FUNCTION_BLOCK FB_InterlockHandler
VAR_INPUT
	i_stInterlockList : ST_InterlockList;
END_VAR
VAR
	s_bInterlocked : BOOL;
	s_sReason : STRING(GVL.g_MAX_LEN_INTERLOCK_REASON);
	i : USINT;
	s_nInterlockCnt : USINT;
	
END_VAR


s_bInterlocked := FALSE;
s_sReason := '';
s_nInterlockCnt := 0;

FOR i := 0 TO (GVL.g_LEN_INTERLOCK_LIST-1) DO
	IF i_stInterlockList.arr_Interlocks[i].bState THEN
		s_bInterlocked := i_stInterlockList.arr_Interlocks[i].bState;
		s_sReason := i_stInterlockList.arr_Interlocks[i].sReason;
		EXIT;
	END_IF
END_FOR

PROPERTY PUBLIC p_bInterlocked : BOOL
GET

p_bInterlocked := s_bInterlocked;
END_GET
END_PROPERTY

PROPERTY PUBLIC p_sReason : STRING
GET

p_sReason := s_sReason;
END_GET
END_PROPERTY

PROPERTY PUBLIC p_stInterlock : ST_Interlock
GET

p_stInterlock.bState := s_bInterlocked;
p_stInterlock.sReason := s_sReason;
END_GET
END_PROPERTY

END_FUNCTION_BLOCK

(* stored: Version 1.1.0.1, ProductVersion 3.1.4024.12
   POU FB_InterlockHandler: Id {3f803ac0-c811-44d7-bc37-de6385932f87}, SpecialFunc None
   Property p_bInterlocked: Id {86e04223-6d35-4c0b-a8e3-7fa2c5ae859f}
   Get Get: Id {18a6c684-2c70-43a4-813f-00bd04500324}
   Property p_sReason: Id {aaf90641-7dc3-4684-ad11-173ff784777c}
   Get Get: Id {dcfe3acf-6a85-4f02-8995-d2803f5f511d}
   Property p_stInterlock: Id {6c20b4ab-4661-4715-b2e6-31a8d7320398}
   Get Get: Id {0fc47193-ceb4-4c97-976e-4185eb439179} *)
